$TOOL = {FRAME: X 0.000,Y 0.000,Z 10.000,A 0.000,B 0.000,C 0.000}
; $TOOL = TOOL_DATA[1]
; --------------------------
PTP {A1 -82.95030,A2 -64.67180,A3 114.28100,A4 38.73570,A5 -58.51180,A6 -21.16620}
; ---- Setting reference (Base) ----
$BASE = {FRAME: X 0.000,Y 0.000,Z 0.000,A 0.000,B 0.000,C 0.000}
; --------------------------
; ---- Setting tool (TCP) ----
; TOOL_DATA[1] = {FRAME: X 0.000,Y 0.000,Z 10.000,A 0.000,B 0.000,C 0.000}
$TOOL = {FRAME: X 0.000,Y 0.000,Z 10.000,A 0.000,B 0.000,C 0.000}
; $TOOL = TOOL_DATA[1]
; --------------------------
PTP {A1 -88.03700,A2 -65.67870,A3 116.47500,A4 -3.49437,A5 -53.88260,A6 3.65705}
; ---- Setting reference (Base) ----
$BASE = {FRAME: X 0.000,Y 0.000,Z 0.000,A 0.000,B 0.000,C 0.000}
; --------------------------
; ---- Setting tool (TCP) ----
; TOOL_DATA[1] = {FRAME: X 0.000,Y 0.000,Z 10.000,A 0.000,B 0.000,C 0.000}
$TOOL = {FRAME: X 0.000,Y 0.000,Z 10.000,A 0.000,B 0.000,C 0.000}
; $TOOL = TOOL_DATA[1]
; --------------------------
PTP {A1 -88.03700,A2 -65.67870,A3 116.47500,A4 -3.49437,A5 -53.88260,A6 -26.34300}
; ---- Setting reference (Base) ----
$BASE = {FRAME: X 0.000,Y 0.000,Z 0.000,A 0.000,B 0.000,C 0.000}
; --------------------------
; ---- Setting tool (TCP) ----
; TOOL_DATA[1] = {FRAME: X 0.000,Y 0.000,Z 10.000,A 0.000,B 0.000,C 0.000}
$TOOL = {FRAME: X 0.000,Y 0.000,Z 10.000,A 0.000,B 0.000,C 0.000}
; $TOOL = TOOL_DATA[1]
; --------------------------
PTP {A1 -88.03700,A2 -65.67870,A3 116.47500,A4 -3.49437,A5 -53.88260,A6 33.65700}
; ---- Setting reference (Base) ----
$BASE = {FRAME: X 0.000,Y 0.000,Z 0.000,A 0.000,B 0.000,C 0.000}
; --------------------------
; ---- Setting tool (TCP) ----
; TOOL_DATA[1] = {FRAME: X 0.000,Y 0.000,Z 10.000,A 0.000,B 0.000,C 0.000}
$TOOL = {FRAME: X 0.000,Y 0.000,Z 10.000,A 0.000,B 0.000,C 0.000}
; $TOOL = TOOL_DATA[1]
; --------------------------
PTP {A1 -88.03700,A2 -65.67870,A3 116.47500,A4 -3.49437,A5 -53.88260,A6 3.65705}
; ---- Setting reference (Base) ----
$BASE = {FRAME: X 0.000,Y 0.000,Z 0.000,A 0.000,B 0.000,C 0.000}
; --------------------------
; ---- Setting tool (TCP) ----
; TOOL_DATA[1] = {FRAME: X 0.000,Y 0.000,Z 10.000,A 0.000,B 0.000,C 0.000}
$TOOL = {FRAME: X 0.000,Y 0.000,Z 10.000,A 0.000,B 0.000,C 0.000}
; $TOOL = TOOL_DATA[1]
; --------------------------
PTP {A1 -89.25720,A2 -65.56940,A3 116.36100,A4 -5.00091,A5 -53.93510,A6 4.60935}
; ---- Setting reference (Base) ----
$BASE = {FRAME: X 0.000,Y 0.000,Z 0.000,A 0.000,B 0.000,C 0.000}
; --------------------------
; ---- Setting tool (TCP) ----
; TOOL_DATA[1] = {FRAME: X 0.000,Y 0.000,Z 10.000,A 0.000,B 0.000,C 0.000}
$TOOL = {FRAME: X 0.000,Y 0.000,Z 10.000,A 0.000,B 0.000,C 0.000}
; $TOOL = TOOL_DATA[1]
; --------------------------
PTP {A1 -94.11860,A2 -63.67460,A3 113.22500,A4 -44.95250,A5 -62.66360,A6 27.06740}
; ---- Setting reference (Base) ----
$BASE = {FRAME: X 0.000,Y 0.000,Z 0.000,A 0.000,B 0.000,C 0.000}
; --------------------------
; ---- Setting tool (TCP) ----
; TOOL_DATA[1] = {FRAME: X 0.000,Y 0.000,Z 10.000,A 0.000,B 0.000,C 0.000}
$TOOL = {FRAME: X 0.000,Y 0.000,Z 10.000,A 0.000,B 0.000,C 0.000}
; $TOOL = TOOL_DATA[1]
; --------------------------
PTP {A1 -84.14550,A2 -64.66570,A3 114.34200,A4 37.42330,A5 -58.08690,A6 -20.40190}
; ---- Setting reference (Base) ----
$BASE = {FRAME: X 0.000,Y 0.000,Z 0.000,A 0.000,B 0.000,C 0.000}
; --------------------------
; ---- Setting tool (TCP) ----
; TOOL_DATA[1] = {FRAME: X 0.000,Y 0.000,Z 10.000,A 0.000,B 0.000,C 0.000}
$TOOL = {FRAME: X 0.000,Y 0.000,Z 10.000,A 0.000,B 0.000,C 0.000}
; $TOOL = TOOL_DATA[1]
; --------------------------
PTP {A1 -89.25720,A2 -65.56940,A3 116.36100,A4 -5.00091,A5 -53.93510,A6 4.60935}
; ---- Setting reference (Base) ----
$BASE = {FRAME: X 0.000,Y 0.000,Z 0.000,A 0.000,B 0.000,C 0.000}
; --------------------------
; ---- Setting tool (TCP) ----
; TOOL_DATA[1] = {FRAME: X 0.000,Y 0.000,Z 10.000,A 0.000,B 0.000,C 0.000}
$TOOL = {FRAME: X 0.000,Y 0.000,Z 10.000,A 0.000,B 0.000,C 0.000}
; $TOOL = TOOL_DATA[1]
; --------------------------
PTP {A1 -89.25720,A2 -65.56940,A3 116.36100,A4 -5.00091,A5 -53.93510,A6 -25.39060}
; ---- Setting reference (Base) ----
$BASE = {FRAME: X 0.000,Y 0.000,Z 0.000,A 0.000,B 0.000,C 0.000}
; --------------------------
; ---- Setting tool (TCP) ----
; TOOL_DATA[1] = {FRAME: X 0.000,Y 0.000,Z 10.000,A 0.000,B 0.000,C 0.000}
$TOOL = {FRAME: X 0.000,Y 0.000,Z 10.000,A 0.000,B 0.000,C 0.000}
; $TOOL = TOOL_DATA[1]
; --------------------------
PTP {A1 -89.25720,A2 -65.56940,A3 116.36100,A4 -5.00091,A5 -53.93510,A6 34.60940}
; ---- Setting reference (Base) ----
$BASE = {FRAME: X 0.000,Y 0.000,Z 0.000,A 0.000,B 0.000,C 0.000}
; --------------------------
; ---- Setting tool (TCP) ----
; TOOL_DATA[1] = {FRAME: X 0.000,Y 0.000,Z 10.000,A 0.000,B 0.000,C 0.000}
$TOOL = {FRAME: X 0.000,Y 0.000,Z 10.000,A 0.000,B 0.000,C 0.000}
; $TOOL = TOOL_DATA[1]
; --------------------------
PTP {A1 -89.25720,A2 -65.56940,A3 116.36100,A4 -5.00091,A5 -53.93510,A6 4.60935}
; ---- Setting reference (Base) ----
$BASE = {FRAME: X 0.000,Y 0.000,Z 0.000,A 0.000,B 0.000,C 0.000}
; --------------------------
; ---- Setting tool (TCP) ----
; TOOL_DATA[1] = {FRAME: X 0.000,Y 0.000,Z 10.000,A 0.000,B 0.000,C 0.000}
$TOOL = {FRAME: X 0.000,Y 0.000,Z 10.000,A 0.000,B 0.000,C 0.000}
; $TOOL = TOOL_DATA[1]
; --------------------------
PTP {A1 -90.47370,A2 -65.43600,A3 116.20600,A4 -6.50179,A5 -53.99030,A6 5.55851}
; ---- Setting reference (Base) ----
$BASE = {FRAME: X 0.000,Y 0.000,Z 0.000,A 0.000,B 0.000,C 0.000}
; --------------------------
; ---- Setting tool (TCP) ----
; TOOL_DATA[1] = {FRAME: X 0.000,Y 0.000,Z 10.000,A 0.000,B 0.000,C 0.000}
$TOOL = {FRAME: X 0.000,Y 0.000,Z 10.000,A 0.000,B 0.000,C 0.000}
; $TOOL = TOOL_DATA[1]
; --------------------------
PTP {A1 -95.28170,A2 -63.44730,A3 112.90000,A4 -46.14340,A5 -63.13430,A6 27.74000}
; ---- Setting reference (Base) ----
$BASE = {FRAME: X 0.000,Y 0.000,Z 0.000,A 0.000,B 0.000,C 0.000}
; --------------------------
; ---- Setting tool (TCP) ----
; TOOL_DATA[1] = {FRAME: X 0.000,Y 0.000,Z 10.000,A 0.000,B 0.000,C 0.000}
$TOOL = {FRAME: X 0.000,Y 0.000,Z 10.000,A 0.000,B 0.000,C 0.000}
; $TOOL = TOOL_DATA[1]
; --------------------------
PTP {A1 -85.34150,A2 -64.63550,A3 114.36100,A4 36.10340,A5 -57.66350,A6 -19.63520}
; ---- Setting reference (Base) ----
$BASE = {FRAME: X 0.000,Y 0.000,Z 0.000,A 0.000,B 0.000,C 0.000}
; --------------------------
; ---- Setting tool (TCP) ----
; TOOL_DATA[1] = {FRAME: X 0.000,Y 0.000,Z 10.000,A 0.000,B 0.000,C 0.000}
$TOOL = {FRAME: X 0.000,Y 0.000,Z 10.000,A 0.000,B 0.000,C 0.000}
; $TOOL = TOOL_DATA[1]
; --------------------------
PTP {A1 -90.47370,A2 -65.43600,A3 116.20600,A4 -6.50179,A5 -53.99030,A6 5.55851}
; ---- Setting reference (Base) ----
$BASE = {FRAME: X 0.000,Y 0.000,Z 0.000,A 0.000,B 0.000,C 0.000}
; --------------------------
; ---- Setting tool (TCP) ----
; TOOL_DATA[1] = {FRAME: X 0.000,Y 0.000,Z 10.000,A 0.000,B 0.000,C 0.000}
$TOOL = {FRAME: X 0.000,Y 0.000,Z 10.000,A 0.000,B 0.000,C 0.000}
; $TOOL = TOOL_DATA[1]
; --------------------------
PTP {A1 -90.47370,A2 -65.43600,A3 116.20600,A4 -6.50179,A5 -53.99030,A6 -24.44150}
; ---- Setting reference (Base) ----
$BASE = {FRAME: X 0.000,Y 0.000,Z 0.000,A 0.000,B 0.000,C 0.000}
; --------------------------
; ---- Setting tool (TCP) ----
; TOOL_DATA[1] = {FRAME: X 0.000,Y 0.000,Z 10.000,A 0.000,B 0.000,C 0.000}
$TOOL = {FRAME: X 0.000,Y 0.000,Z 10.000,A 0.000,B 0.000,C 0.000}
; $TOOL = TOOL_DATA[1]
; --------------------------
PTP {A1 -90.47370,A2 -65.43600,A3 116.20600,A4 -6.50179,A5 -53.99030,A6 35.55850}
; ---- Setting reference (Base) ----
$BASE = {FRAME: X 0.000,Y 0.000,Z 0.000,A 0.000,B 0.000,C 0.000}
; --------------------------
; ---- Setting tool (TCP) ----
; TOOL_DATA[1] = {FRAME: X 0.000,Y 0.000,Z 10.000,A 0.000,B 0.000,C 0.000}
$TOOL = {FRAME: X 0.000,Y 0.000,Z 10.000,A 0.000,B 0.000,C 0.000}
; $TOOL = TOOL_DATA[1]
; --------------------------
PTP {A1 -90.47370,A2 -65.43600,A3 116.20600,A4 -6.50179,A5 -53.99030,A6 5.55851}
; ---- Setting reference (Base) ----
$BASE = {FRAME: X 0.000,Y 0.000,Z 0.000,A 0.000,B 0.000,C 0.000}
; --------------------------
; ---- Setting tool (TCP) ----
; TOOL_DATA[1] = {FRAME: X 0.000,Y 0.000,Z 10.000,A 0.000,B 0.000,C 0.000}
$TOOL = {FRAME: X 0.000,Y 0.000,Z 10.000,A 0.000,B 0.000,C 0.000}
; $TOOL = TOOL_DATA[1]
; --------------------------
PTP {A1 -91.68540,A2 -65.27870,A3 116.00900,A4 -7.99594,A5 -54.04770,A6 6.50451}
; ---- Setting reference (Base) ----
$BASE = {FRAME: X 0.000,Y 0.000,Z 0.000,A 0.000,B 0.000,C 0.000}
; --------------------------
; ---- Setting tool (TCP) ----
; TOOL_DATA[1] = {FRAME: X 0.000,Y 0.000,Z 10.000,A 0.000,B 0.000,C 0.000}
$TOOL = {FRAME: X 0.000,Y 0.000,Z 10.000,A 0.000,B 0.000,C 0.000}
; $TOOL = TOOL_DATA[1]
; --------------------------
PTP {A1 -96.43640,A2 -63.19760,A3 112.53500,A4 -47.32060,A5 -63.60230,A6 28.41040}
; ---- Setting reference (Base) ----
$BASE = {FRAME: X 0.000,Y 0.000,Z 0.000,A 0.000,B 0.000,C 0.000}
; --------------------------
; ---- Setting tool (TCP) ----
; TOOL_DATA[1] = {FRAME: X 0.000,Y 0.000,Z 10.000,A 0.000,B 0.000,C 0.000}
$TOOL = {FRAME: X 0.000,Y 0.000,Z 10.000,A 0.000,B 0.000,C 0.000}
; $TOOL = TOOL_DATA[1]
; --------------------------
PTP {A1 -86.53740,A2 -64.58130,A3 114.33900,A4 34.77700,A5 -57.24160,A6 -18.86620}
; ---- Setting reference (Base) ----
$BASE = {FRAME: X 0.000,Y 0.000,Z 0.000,A 0.000,B 0.000,C 0.000}
; --------------------------
; ---- Setting tool (TCP) ----
; TOOL_DATA[1] = {FRAME: X 0.000,Y 0.000,Z 10.000,A 0.000,B 0.000,C 0.000}
$TOOL = {FRAME: X 0.000,Y 0.000,Z 10.000,A 0.000,B 0.000,C 0.000}
; $TOOL = TOOL_DATA[1]
; --------------------------
PTP {A1 -91.68540,A2 -65.27870,A3 116.00900,A4 -7.99594,A5 -54.04770,A6 6.50451}
; ---- Setting reference (Base) ----
$BASE = {FRAME: X 0.000,Y 0.000,Z 0.000,A 0.000,B 0.000,C 0.000}
; --------------------------
; ---- Setting tool (TCP) ----
; TOOL_DATA[1] = {FRAME: X 0.000,Y 0.000,Z 10.000,A 0.000,B 0.000,C 0.000}
$TOOL = {FRAME: X 0.000,Y 0.000,Z 10.000,A 0.000,B 0.000,C 0.000}
; $TOOL = TOOL_DATA[1]
; --------------------------
PTP {A1 -91.68540,A2 -65.27870,A3 116.00900,A4 -7.99594,A5 -54.04770,A6 -23.49550}
; ---- Setting reference (Base) ----
$BASE = {FRAME: X 0.000,Y 0.000,Z 0.000,A 0.000,B 0.000,C 0.000}
; --------------------------
; ---- Setting tool (TCP) ----
; TOOL_DATA[1] = {FRAME: X 0.000,Y 0.000,Z 10.000,A 0.000,B 0.000,C 0.000}
$TOOL = {FRAME: X 0.000,Y 0.000,Z 10.000,A 0.000,B 0.000,C 0.000}
; $TOOL = TOOL_DATA[1]
; --------------------------
PTP {A1 -91.68540,A2 -65.27870,A3 116.00900,A4 -7.99594,A5 -54.04770,A6 36.50450}
; ---- Setting reference (Base) ----
$BASE = {FRAME: X 0.000,Y 0.000,Z 0.000,A 0.000,B 0.000,C 0.000}
; --------------------------
; ---- Setting tool (TCP) ----
; TOOL_DATA[1] = {FRAME: X 0.000,Y 0.000,Z 10.000,A 0.000,B 0.000,C 0.000}
$TOOL = {FRAME: X 0.000,Y 0.000,Z 10.000,A 0.000,B 0.000,C 0.000}
; $TOOL = TOOL_DATA[1]
; --------------------------
PTP {A1 -91.68540,A2 -65.27870,A3 116.00900,A4 -7.99594,A5 -54.04770,A6 6.50451}
; ---- Setting reference (Base) ----
$BASE = {FRAME: X 0.000,Y 0.000,Z 0.000,A 0.000,B 0.000,C 0.000}
; --------------------------
; ---- Setting tool (TCP) ----
; TOOL_DATA[1] = {FRAME: X 0.000,Y 0.000,Z 10.000,A 0.000,B 0.000,C 0.000}
$TOOL = {FRAME: X 0.000,Y 0.000,Z 10.000,A 0.000,B 0.000,C 0.000}
; $TOOL = TOOL_DATA[1]
; --------------------------
PTP {A1 -92.89120,A2 -65.09770,A3 115.77000,A4 -9.48230,A5 -54.10710,A6 7.44741}
; ---- Setting reference (Base) ----
$BASE = {FRAME: X 0.000,Y 0.000,Z 0.000,A 0.000,B 0.000,C 0.000}
; --------------------------
; ---- Setting tool (TCP) ----
; TOOL_DATA[1] = {FRAME: X 0.000,Y 0.000,Z 10.000,A 0.000,B 0.000,C 0.000}
$TOOL = {FRAME: X 0.000,Y 0.000,Z 10.000,A 0.000,B 0.000,C 0.000}
; $TOOL = TOOL_DATA[1]
; --------------------------
PTP {A1 -97.58180,A2 -62.92570,A3 112.13000,A4 -48.48350,A5 -64.06730,A6 29.07910}
; ---- Setting reference (Base) ----
$BASE = {FRAME: X 0.000,Y 0.000,Z 0.000,A 0.000,B 0.000,C 0.000}
; --------------------------
; ---- Setting tool (TCP) ----
; TOOL_DATA[1] = {FRAME: X 0.000,Y 0.000,Z 10.000,A 0.000,B 0.000,C 0.000}
$TOOL = {FRAME: X 0.000,Y 0.000,Z 10.000,A 0.000,B 0.000,C 0.000}
; $TOOL = TOOL_DATA[1]
; --------------------------
PTP {A1 -87.73200,A2 -64.50320,A3 114.27600,A4 33.44520,A5 -56.82120,A6 -18.09470}
; ---- Setting reference (Base) ----
$BASE = {FRAME: X 0.000,Y 0.000,Z 0.000,A 0.000,B 0.000,C 0.000}
; --------------------------
; ---- Setting tool (TCP) ----
; TOOL_DATA[1] = {FRAME: X 0.000,Y 0.000,Z 10.000,A 0.000,B 0.000,C 0.000}
$TOOL = {FRAME: X 0.000,Y 0.000,Z 10.000,A 0.000,B 0.000,C 0.000}
; $TOOL = TOOL_DATA[1]
; --------------------------
PTP {A1 -92.89120,A2 -65.09770,A3 115.77000,A4 -9.48230,A5 -54.10710,A6 7.44741}
; ---- Setting reference (Base) ----
$BASE = {FRAME: X 0.000,Y 0.000,Z 0.000,A 0.000,B 0.000,C 0.000}
; --------------------------
; ---- Setting tool (TCP) ----
; TOOL_DATA[1] = {FRAME: X 0.000,Y 0.000,Z 10.000,A 0.000,B 0.000,C 0.000}
$TOOL = {FRAME: X 0.000,Y 0.000,Z 10.000,A 0.000,B 0.000,C 0.000}
; $TOOL = TOOL_DATA[1]
; --------------------------
PTP {A1 -92.89120,A2 -65.09770,A3 115.77000,A4 -9.48230,A5 -54.10710,A6 -22.55260}
; ---- Setting reference (Base) ----
$BASE = {FRAME: X 0.000,Y 0.000,Z 0.000,A 0.000,B 0.000,C 0.000}
; --------------------------
; ---- Setting tool (TCP) ----
; TOOL_DATA[1] = {FRAME: X 0.000,Y 0.000,Z 10.000,A 0.000,B 0.000,C 0.000}
$TOOL = {FRAME: X 0.000,Y 0.000,Z 10.000,A 0.000,B 0.000,C 0.000}
; $TOOL = TOOL_DATA[1]
; --------------------------
PTP {A1 -92.89120,A2 -65.09770,A3 115.77000,A4 -9.48230,A5 -54.10710,A6 37.44740}
; ---- Setting reference (Base) ----
$BASE = {FRAME: X 0.000,Y 0.000,Z 0.000,A 0.000,B 0.000,C 0.000}
; --------------------------
; ---- Setting tool (TCP) ----
; TOOL_DATA[1] = {FRAME: X 0.000,Y 0.000,Z 10.000,A 0.000,B 0.000,C 0.000}
$TOOL = {FRAME: X 0.000,Y 0.000,Z 10.000,A 0.000,B 0.000,C 0.000}
; $TOOL = TOOL_DATA[1]
; --------------------------
PTP {A1 -92.89120,A2 -65.09770,A3 115.77000,A4 -9.48230,A5 -54.10710,A6 7.44741}
; ---- Setting reference (Base) ----
$BASE = {FRAME: X 0.000,Y 0.000,Z 0.000,A 0.000,B 0.000,C 0.000}
; --------------------------
; ---- Setting tool (TCP) ----
; TOOL_DATA[1] = {FRAME: X 0.000,Y 0.000,Z 10.000,A 0.000,B 0.000,C 0.000}
$TOOL = {FRAME: X 0.000,Y 0.000,Z 10.000,A 0.000,B 0.000,C 0.000}
; $TOOL = TOOL_DATA[1]
; --------------------------
PTP {A1 -94.09020,A2 -64.89330,A3 115.49100,A4 -10.95990,A5 -54.16820,A6 8.38728}
; ---- Setting reference (Base) ----
$BASE = {FRAME: X 0.000,Y 0.000,Z 0.000,A 0.000,B 0.000,C 0.000}
; --------------------------
; ---- Setting tool (TCP) ----
; TOOL_DATA[1] = {FRAME: X 0.000,Y 0.000,Z 10.000,A 0.000,B 0.000,C 0.000}
$TOOL = {FRAME: X 0.000,Y 0.000,Z 10.000,A 0.000,B 0.000,C 0.000}
; $TOOL = TOOL_DATA[1]
; --------------------------
PTP {A1 -98.71720,A2 -62.63190,A3 111.68400,A4 -49.63160,A5 -64.52910,A6 29.74660}
; ---- Setting reference (Base) ----
$BASE = {FRAME: X 0.000,Y 0.000,Z 0.000,A 0.000,B 0.000,C 0.000}
; --------------------------
; ---- Setting tool (TCP) ----
; TOOL_DATA[1] = {FRAME: X 0.000,Y 0.000,Z 10.000,A 0.000,B 0.000,C 0.000}
$TOOL = {FRAME: X 0.000,Y 0.000,Z 10.000,A 0.000,B 0.000,C 0.000}
; $TOOL = TOOL_DATA[1]
; --------------------------
PTP {A1 -88.92440,A2 -64.40130,A3 114.17200,A4 32.10900,A5 -56.40220,A6 -17.32090}
; ---- Setting reference (Base) ----
$BASE = {FRAME: X 0.000,Y 0.000,Z 0.000,A 0.000,B 0.000,C 0.000}
; --------------------------
; ---- Setting tool (TCP) ----
; TOOL_DATA[1] = {FRAME: X 0.000,Y 0.000,Z 10.000,A 0.000,B 0.000,C 0.000}
$TOOL = {FRAME: X 0.000,Y 0.000,Z 10.000,A 0.000,B 0.000,C 0.000}
; $TOOL = TOOL_DATA[1]
; --------------------------
PTP {A1 -94.09020,A2 -64.89330,A3 115.49100,A4 -10.95990,A5 -54.16820,A6 8.38728}
; ---- Setting reference (Base) ----
$BASE = {FRAME: X 0.000,Y 0.000,Z 0.000,A 0.000,B 0.000,C 0.000}
; --------------------------
; ---- Setting tool (TCP) ----
; TOOL_DATA[1] = {FRAME: X 0.000,Y 0.000,Z 10.000,A 0.000,B 0.000,C 0.000}
$TOOL = {FRAME: X 0.000,Y 0.000,Z 10.000,A 0.000,B 0.000,C 0.000}
; $TOOL = TOOL_DATA[1]
; --------------------------
PTP {A1 -94.09020,A2 -64.89330,A3 115.49100,A4 -10.95990,A5 -54.16820,A6 -21.61270}
; ---- Setting reference (Base) ----
$BASE = {FRAME: X 0.000,Y 0.000,Z 0.000,A 0.000,B 0.000,C 0.000}
; --------------------------
; ---- Setting tool (TCP) ----
; TOOL_DATA[1] = {FRAME: X 0.000,Y 0.000,Z 10.000,A 0.000,B 0.000,C 0.000}
$TOOL = {FRAME: X 0.000,Y 0.000,Z 10.000,A 0.000,B 0.000,C 0.000}
; $TOOL = TOOL_DATA[1]
; --------------------------
PTP {A1 -94.09020,A2 -64.89330,A3 115.49100,A4 -10.95990,A5 -54.16820,A6 38.38730}
; ---- Setting reference (Base) ----
$BASE = {FRAME: X 0.000,Y 0.000,Z 0.000,A 0.000,B 0.000,C 0.000}
; --------------------------
; ---- Setting tool (TCP) ----
; TOOL_DATA[1] = {FRAME: X 0.000,Y 0.000,Z 10.000,A 0.000,B 0.000,C 0.000}
$TOOL = {FRAME: X 0.000,Y 0.000,Z 10.000,A 0.000,B 0.000,C 0.000}
; $TOOL = TOOL_DATA[1]
; --------------------------
PTP {A1 -94.09020,A2 -64.89330,A3 115.49100,A4 -10.95990,A5 -54.16820,A6 8.38728}
; ---- Setting reference (Base) ----
$BASE = {FRAME: X 0.000,Y 0.000,Z 0.000,A 0.000,B 0.000,C 0.000}
; --------------------------
; ---- Setting tool (TCP) ----
; TOOL_DATA[1] = {FRAME: X 0.000,Y 0.000,Z 10.000,A 0.000,B 0.000,C 0.000}
$TOOL = {FRAME: X 0.000,Y 0.000,Z 10.000,A 0.000,B 0.000,C 0.000}
; $TOOL = TOOL_DATA[1]
; --------------------------
PTP {A1 -95.28130,A2 -64.66580,A3 115.17100,A4 -12.42780,A5 -54.23060,A6 9.32425}
; ---- Setting reference (Base) ----
$BASE = {FRAME: X 0.000,Y 0.000,Z 0.000,A 0.000,B 0.000,C 0.000}
; --------------------------
; ---- Setting tool (TCP) ----
; TOOL_DATA[1] = {FRAME: X 0.000,Y 0.000,Z 10.000,A 0.000,B 0.000,C 0.000}
$TOOL = {FRAME: X 0.000,Y 0.000,Z 10.000,A 0.000,B 0.000,C 0.000}
; $TOOL = TOOL_DATA[1]
; --------------------------
PTP {A1 -99.84190,A2 -62.31650,A3 111.19900,A4 -50.76430,A5 -64.98760,A6 30.41350}
; ---- Setting reference (Base) ----
$BASE = {FRAME: X 0.000,Y 0.000,Z 0.000,A 0.000,B 0.000,C 0.000}
; --------------------------
; ---- Setting tool (TCP) ----
; TOOL_DATA[1] = {FRAME: X 0.000,Y 0.000,Z 10.000,A 0.000,B 0.000,C 0.000}
$TOOL = {FRAME: X 0.000,Y 0.000,Z 10.000,A 0.000,B 0.000,C 0.000}
; $TOOL = TOOL_DATA[1]
; --------------------------
PTP {A1 -90.11350,A2 -64.27580,A3 114.02600,A4 30.76930,A5 -55.98450,A6 -16.54460}
; ---- Setting reference (Base) ----
$BASE = {FRAME: X 0.000,Y 0.000,Z 0.000,A 0.000,B 0.000,C 0.000}
; --------------------------
; ---- Setting tool (TCP) ----
; TOOL_DATA[1] = {FRAME: X 0.000,Y 0.000,Z 10.000,A 0.000,B 0.000,C 0.000}
$TOOL = {FRAME: X 0.000,Y 0.000,Z 10.000,A 0.000,B 0.000,C 0.000}
; $TOOL = TOOL_DATA[1]
; --------------------------
PTP {A1 -95.28130,A2 -64.66580,A3 115.17100,A4 -12.42780,A5 -54.23060,A6 9.32425}
; ---- Setting reference (Base) ----
$BASE = {FRAME: X 0.000,Y 0.000,Z 0.000,A 0.000,B 0.000,C 0.000}
; --------------------------
; ---- Setting tool (TCP) ----
; TOOL_DATA[1] = {FRAME: X 0.000,Y 0.000,Z 10.000,A 0.000,B 0.000,C 0.000}
$TOOL = {FRAME: X 0.000,Y 0.000,Z 10.000,A 0.000,B 0.000,C 0.000}
; $TOOL = TOOL_DATA[1]
; --------------------------
PTP {A1 -95.28130,A2 -64.66580,A3 115.17100,A4 -12.42780,A5 -54.23060,A6 -20.67570}
; ---- Setting reference (Base) ----
$BASE = {FRAME: X 0.000,Y 0.000,Z 0.000,A 0.000,B 0.000,C 0.000}
; --------------------------
; ---- Setting tool (TCP) ----
; TOOL_DATA[1] = {FRAME: X 0.000,Y 0.000,Z 10.000,A 0.000,B 0.000,C 0.000}
$TOOL = {FRAME: X 0.000,Y 0.000,Z 10.000,A 0.000,B 0.000,C 0.000}
; $TOOL = TOOL_DATA[1]
; --------------------------
PTP {A1 -95.28130,A2 -64.66580,A3 115.17100,A4 -12.42780,A5 -54.23060,A6 39.32430}
; ---- Setting reference (Base) ----
$BASE = {FRAME: X 0.000,Y 0.000,Z 0.000,A 0.000,B 0.000,C 0.000}
; --------------------------
; ---- Setting tool (TCP) ----
; TOOL_DATA[1] = {FRAME: X 0.000,Y 0.000,Z 10.000,A 0.000,B 0.000,C 0.000}
$TOOL = {FRAME: X 0.000,Y 0.000,Z 10.000,A 0.000,B 0.000,C 0.000}
; $TOOL = TOOL_DATA[1]
; --------------------------
PTP {A1 -95.28130,A2 -64.66580,A3 115.17100,A4 -12.42780,A5 -54.23060,A6 9.32425}
; ---- Setting reference (Base) ----
$BASE = {FRAME: X 0.000,Y 0.000,Z 0.000,A 0.000,B 0.000,C 0.000}
; --------------------------
; ---- Setting tool (TCP) ----
; TOOL_DATA[1] = {FRAME: X 0.000,Y 0.000,Z 10.000,A 0.000,B 0.000,C 0.000}
$TOOL = {FRAME: X 0.000,Y 0.000,Z 10.000,A 0.000,B 0.000,C 0.000}
; $TOOL = TOOL_DATA[1]
; --------------------------
PTP {A1 -96.46360,A2 -64.41550,A3 114.80900,A4 -13.88510,A5 -54.29400,A6 10.25850}
; ---- Setting reference (Base) ----
$BASE = {FRAME: X 0.000,Y 0.000,Z 0.000,A 0.000,B 0.000,C 0.000}
; --------------------------
; ---- Setting tool (TCP) ----
; TOOL_DATA[1] = {FRAME: X 0.000,Y 0.000,Z 10.000,A 0.000,B 0.000,C 0.000}
$TOOL = {FRAME: X 0.000,Y 0.000,Z 10.000,A 0.000,B 0.000,C 0.000}
; $TOOL = TOOL_DATA[1]
; --------------------------
PTP {A1 -100.95500,A2 -61.97980,A3 110.67400,A4 -51.88120,A5 -65.44260,A6 31.08010}
; ---- Setting reference (Base) ----
$BASE = {FRAME: X 0.000,Y 0.000,Z 0.000,A 0.000,B 0.000,C 0.000}
; --------------------------
; ---- Setting tool (TCP) ----
; TOOL_DATA[1] = {FRAME: X 0.000,Y 0.000,Z 10.000,A 0.000,B 0.000,C 0.000}
$TOOL = {FRAME: X 0.000,Y 0.000,Z 10.000,A 0.000,B 0.000,C 0.000}
; $TOOL = TOOL_DATA[1]
; --------------------------
PTP {A1 -91.29840,A2 -64.12680,A3 113.84000,A4 29.42740,A5 -55.56810,A6 -15.76600}
; ---- Setting reference (Base) ----
$BASE = {FRAME: X 0.000,Y 0.000,Z 0.000,A 0.000,B 0.000,C 0.000}
; --------------------------
; ---- Setting tool (TCP) ----
; TOOL_DATA[1] = {FRAME: X 0.000,Y 0.000,Z 10.000,A 0.000,B 0.000,C 0.000}
$TOOL = {FRAME: X 0.000,Y 0.000,Z 10.000,A 0.000,B 0.000,C 0.000}
; $TOOL = TOOL_DATA[1]
; --------------------------
PTP {A1 -96.46360,A2 -64.41550,A3 114.80900,A4 -13.88510,A5 -54.29400,A6 10.25850}
; ---- Setting reference (Base) ----
$BASE = {FRAME: X 0.000,Y 0.000,Z 0.000,A 0.000,B 0.000,C 0.000}
; --------------------------
; ---- Setting tool (TCP) ----
; TOOL_DATA[1] = {FRAME: X 0.000,Y 0.000,Z 10.000,A 0.000,B 0.000,C 0.000}
$TOOL = {FRAME: X 0.000,Y 0.000,Z 10.000,A 0.000,B 0.000,C 0.000}

; Continue running program as cascaded execution
Kuka_Relative_Mo1()

END
